Universal Robots PolyScope program: get-movement.urp

Program get-movement (installation=default directory=/ursim/programs createdIn=3.15.8.106339 lastSavedIn=3.15.8.106339 robotSerialNumber=2018359999)
Calibrated DH parameters: a=[0, -0.425, -0.39225, 0, 0, 0]; d=[0.089159, 0, 0, 0.10915, 0.09465, 0.0823]; alpha=[1.570796, 0, 0, 1.570796, -1.570796, 0]; deltaTheta=[0, 0, 0, 0, 0, 0]
BeforeStart
  MoveJ speed 60 deg/s, acceleration 80 deg/s^2 (useActiveTCP=true)
    Waypoint Waypoint_1: TCP in base x=474.55 y=-109.15 z=608.809 mm, rx=-1.2092 ry=1.2092 rz=-1.2092 rad; joints [0, -90, -90, 0, 90, 0] deg
  setp := p[0,0,0,0,0,0]
  movement := False
Robot Program (runOnlyOnce=false)
  If setp ≟p[0,0,0,0,0,0]
    movement := False
  ElseIf setp[0] == 0 and setp[1] == 0 and setp[2] == 0
    movement := False
  Else 
    movement := True
  If movement
    MoveL speed 250 mm/s, acceleration 1200 mm/s^2 (useActiveTCP=false) tcp=TCP; feature=Base
      Waypoint Waypoint (Variable): variable=setp
  Script: sync()
Thread Thread_1 (runOnlyOnce=false)
  tmp := p[0,0,0,0,0,0]
  Script: tmp[0]=read_input_float_register(0)
  Script: tmp[1]=read_input_float_register(1)
  Script: tmp[2]=read_input_float_register(2)
  Script: tmp[3]=read_input_float_register(3)
  Script: tmp[4]=read_input_float_register(4)
  Script: tmp[5]=read_input_float_register(5)
  setp := tmp
  Script: sync()
